// TIA Portal V17 export
// export: Created 2021-11-12T21:16:16.1027334Z, ExportSetting WithDefaults, DisplayName Totally Integrated Automation Portal, DisplayVersion V17 Update 1, DisplayName TIA Portal Openness, DisplayVersion V17 Update 1, DisplayName TIA Portal Version Control Interface, DisplayVersion V17, DisplayName SINAMICS Startdrive Advanced, DisplayVersion V17 Update1, DisplayName SINAMICS Startdrive G110M, G120, G120C, G120D, G120P, G115D, DisplayVersion V17 Update1, DisplayName SINAMICS Startdrive G130, G150, S120, S150, SINAMICS MV, S210, DisplayVersion V17 Update1, DisplayName STEP 7 Professional, DisplayVersion V17 Update 1, DisplayName STEP 7 Safety, DisplayVersion V17, DisplayName WinCC Advanced, DisplayVersion V17 Update 1
DATA_BLOCK "DB - 1 - Dados Inversor MB-01"   // DB230
{ S7_Optimized_Access := 'FALSE' }
VERSION : 0.1
// stored: AutoNumber false, IsOnlyStoredInLoadMemory false, IsWriteProtectedInAS false
   VAR RETAIN
      RW_TCPModBUS_IP_Oct_1_MB : USInt := 0;   // IP Octeto 1 do Inversor MB
      RW_TCPModBUS_IP_Oct_2_MB : USInt := 0;   // IP Octeto 2 do Inversor MB
      RW_TCPModBUS_IP_Oct_3_MB : USInt := 0;   // IP Octeto 3 do Inversor MB
      RW_TCPModBUS_IP_Oct_4_MB : USInt := 0;   // IP Octeto 4 do Inversor MB
      RW_MinMotorFreqHz_MB_Hz : UInt := 300;   // Frequência Minima do Motor Utilizado para o controle de velocidade
      RW_MaxMotorFreqHz_MB_Hz : UInt := 600;   // Frequência Máxima do Motor
      RO_SomatorioConsumo_kWh { ExternalAccessible := 'False'; ExternalVisible := 'False'; ExternalWritable := 'False'} : Real;
      RO_CorrenteAtual_A { ExternalAccessible := 'False'; ExternalVisible := 'False'; ExternalWritable := 'False'} : Real;
      RO_FrequenciaAtual_Hz { ExternalAccessible := 'False'; ExternalVisible := 'False'; ExternalWritable := 'False'} : Real;
      RO_PotenciaAtual_kW { ExternalAccessible := 'False'; ExternalVisible := 'False'; ExternalWritable := 'False'} : Real;
      RO_TensaoAtualSaida_V { ExternalVisible := 'False'} : Real;
      RO_MotorRPM { ExternalAccessible := 'False'; ExternalVisible := 'False'; ExternalWritable := 'False'} : Real;
      RO_TempDriveDissipadorCalor_C { ExternalAccessible := 'False'; ExternalVisible := 'False'; ExternalWritable := 'False'} : Real;
      RO_TempDriveCartaoControle_C { ExternalAccessible := 'False'; ExternalVisible := 'False'; ExternalWritable := 'False'} : Real;
      RO_HorimetroMotor_H : Real;
      RO_HorimetroDrive_H : Real;
      RO_UltimoAlarme : Int;
      "RO_AnalogInput53_ma-V" : Real;
      "RO_AnalogInput54_ma-V" : Real;
      Cfg_Potencia_Motor_kW : Real;
      Cfg_Motor_hp : Real;
      Cfg_Motor_TensaoNominal_V : Real;
      Cfg_Corrente_Nominal_A : Real;
      Cfg_Velocidade_Nominal_RPM : Real;
      RO_Numero_de_PartidasMotor : Real;
      RO_Numero_de_PartidasDrive : Real;
      RO_TensaoBarramentoDC_V : Real;
      RO_TensaoAmpla_V : Real;
   END_VAR
BEGIN
END_DATA_BLOCK
